// TIA Portal V17 export
// export: Created 2025-06-26T07:49:44.1812717Z, ExportSetting WithDefaults, DisplayName Totally Integrated Automation Portal, DisplayVersion V17 Update 8, DisplayName TIA Portal Openness, DisplayVersion V17 Update 8, DisplayName TIA Portal Version Control Interface, DisplayVersion V17, DisplayName STEP 7 Professional, DisplayVersion V17 Update 8, DisplayName STEP 7 Safety, DisplayVersion V17 Update 6, DisplayName WinCC Advanced, DisplayVersion V17 Update 8
FUNCTION_BLOCK "fbProcessValve2_V2"   // FB67, FBD
TITLE = Process valve control
{ S7_Optimized_Access := 'TRUE' }
AUTHOR : Heaten
VERSION : 1.0
// stored: AutoNumber true, IsIECCheckEnabled false, IsRetainMemResEnabled false, MemoryReserve 0, SetENOAutomatically false, UDAEnableTagReadback false
   VAR_INPUT
      bOpenReq : Bool;   // 1 = open valve, 0 = do not open valve (Level signal)
      bCloseReq : Bool;   // 1 = close valve, 0 = do not close valve (Level signal)
      bOpenStat : Bool;   // 1 = valve is open, 0 = valve is not open
      bClosedStat : Bool;   // 1 = valve is closed, 0 = valve is not closed
   END_VAR
   VAR_OUTPUT
      bOpenCmd : Bool;
      bCloseCmd : Bool;
   END_VAR
   VAR_IN_OUT
      sTag : "stProcessValve2";
   END_VAR
   VAR
      OpenTimer : TON_TIME;
      CloseTimer { S7_SetPoint := 'True'} : TON_TIME;
   END_VAR
   VAR_TEMP
      Opening : Bool;
      Closing : Bool;
      OpenError : Bool;
      CloseError : Bool;
      OpenReq : Bool;
      CloseReq : Bool;
   END_VAR
   VAR CONSTANT
      STATE_UNKNOWN : USInt := 0;
      STATE_CLOSED : USInt := 1;
      STATE_OPEN : USInt := 2;
      STATE_CLOSING : USInt := 3;
      STATE_OPENING : USInt := 4;
      STATE_CLOSE_ERROR : USInt := 5;
      STATE_OPEN_ERROR : USInt := 6;
   END_VAR
BEGIN

REGION Network 1 (SCL): Description & version history
   // Remember to update the version in the block properties!
   // Process valve control with decoupled states
   // - valve state is directly represented by the feedback
   // - requests are level signals
   // - valve commands are conditions and not states
   // - errors are conditions and not states
   // - different concerns are decoupled: valve state, request & command, error detection
   // - needs no initial state detection or special handling if valve position feedback disappears

   // V1.0.0.0 08.03.2025 HEATEN
   // - Initial version
END_REGION

REGION Network 2: Open Request
   // Choose between auto & manual
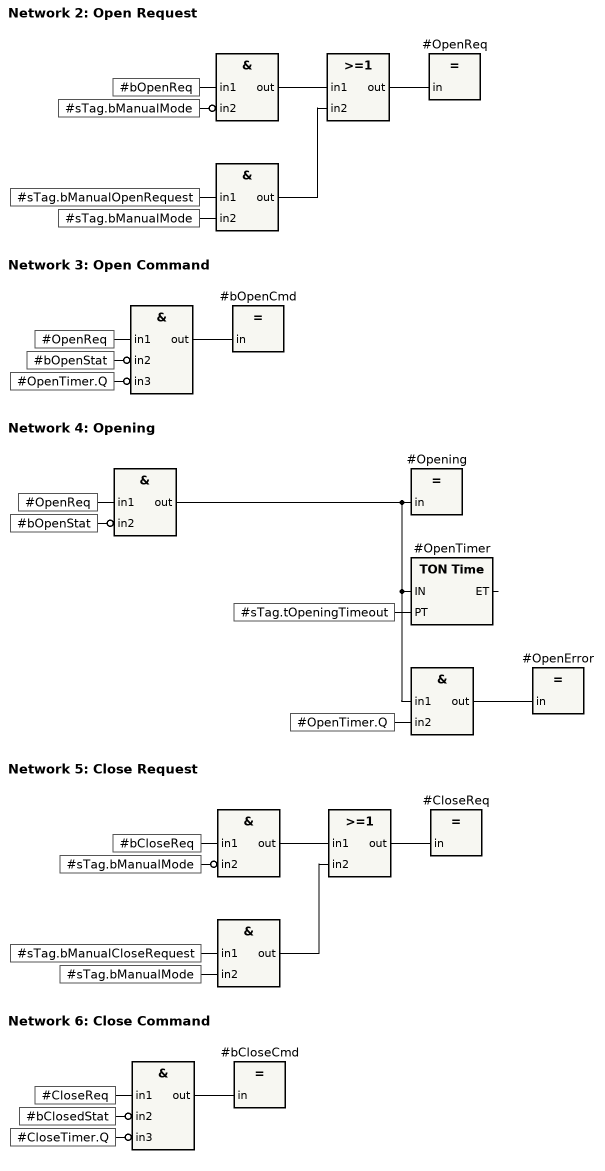
   #OpenReq := (#bOpenReq AND NOT #sTag.bManualMode) OR (#sTag.bManualOpenRequest AND #sTag.bManualMode);
END_REGION

REGION Network 3: Open Command
   // Send the command when the request to open is given
   // Stop when the open status is received or timoeut has occurred
   #bOpenCmd := #OpenReq AND NOT #bOpenStat AND NOT #OpenTimer.Q;
END_REGION

REGION Network 4: Opening
   // Opening as long as the open request is given and no open status received
   // Open timer fires when the request to open doesn't result in an open status after the timeout period
   // Open error active when opening and timeout occurs. Clears when the request is withdrawn or open status received
   #Opening := #OpenReq AND NOT #bOpenStat;
   #OpenTimer(IN := #Opening, PT := #sTag.tOpeningTimeout);   // TON
   #OpenError := #Opening AND #OpenTimer.Q;
END_REGION

REGION Network 5: Close Request
   // Choose between auto & manual
   #CloseReq := (#bCloseReq AND NOT #sTag.bManualMode) OR (#sTag.bManualCloseRequest AND #sTag.bManualMode);
END_REGION

REGION Network 6: Close Command
   // Send the command when the request to close is given
   // Stop when the closed status is received or timoeut has occurred
   #bCloseCmd := #CloseReq AND NOT #bClosedStat AND NOT #CloseTimer.Q;
END_REGION

REGION Network 7: Closing
   // Closing as long as the close request is given and no closed status received
   // Close Timer fires when the request to close doesn't result in a closed status after the timeout period
   // Close error active when closing and timeout occurs. Clears when the request is withdrawn or closed status received
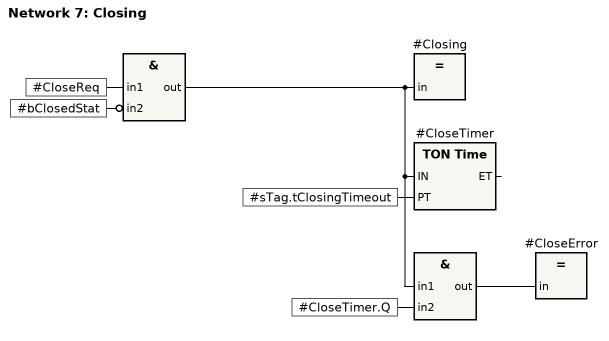
   #Closing := #CloseReq AND NOT #bClosedStat;
   #CloseTimer(IN := #Closing, PT := #sTag.tClosingTimeout);   // TON
   #CloseError := #Closing AND #CloseTimer.Q;
END_REGION

REGION Network 8 (SCL): State representation
   // The order is important, otherwise some conditions are never detected
   IF #OpenError = TRUE THEN
       #sTag.nState := #STATE_OPEN_ERROR;
   ELSIF #CloseError = TRUE THEN
       #sTag.nState := #STATE_CLOSE_ERROR;
   ELSIF #Opening = TRUE THEN
       #sTag.nState := #STATE_OPENING;
   ELSIF #Closing = TRUE THEN
       #sTag.nState := #STATE_CLOSING;
   ELSIF #bOpenStat = TRUE THEN
       #sTag.nState := #STATE_OPEN;
   ELSIF #bClosedStat = TRUE THEN
       #sTag.nState := #STATE_CLOSED;
   ELSE
       #sTag.nState := #STATE_UNKNOWN;
   END_IF;
END_REGION

REGION Network 9 (SCL): Mirror in HMI
   #sTag.bOpenRequest := #OpenReq;
   #sTag.bCloseRequest := #CloseReq;
   #sTag.bOpenStatus := #bOpenStat;
   #sTag.bClosedStatus := #bClosedStat;
   #sTag.bOpenCommand := #bOpenCmd;
   #sTag.bCloseCommand := #bCloseCmd;
END_REGION
END_FUNCTION_BLOCK
